TYPE EL1008IO_typ:
STRUCT
	Input AT %I*: ARRAY[1..8] OF BOOL;
END_STRUCT
END_TYPE

(* stored: Version 1.1.0.1, ProductVersion 3.1.4024.12
   DUT EL1008IO_typ: Id {48959ce0-bbda-01ca-110d-2b36ef8500a7} *)
